# EPICS alarm handler configuration: apps/alhConfig/ecal.alhConfig
#===============================================================================
# ECAL Alarm Config
#===============================================================================

GROUP NULL ECAL

#=======================================
# Subsystems
#=======================================

INCLUDE ECAL /usr/clas12/hps/prod/apps/alhConfig/hv.alhConfig
#INCLUDE ECAL /usr/clas12/hps/prod/apps/alhConfig/ecallv.alhConfig
INCLUDE ECAL /usr/clas12/hps/prod/apps/alhConfig/tempSens.alhConfig
INCLUDE ECAL /usr/clas12/hps/prod/apps/alhConfig/chiller.alhConfig
